(* IEC 61131-3 sources: json/test/String, 1 file *)

(* ---- TestJsonString.st ---- *)
USING AxUnit.Assert;
USING System.Strings;
USING Simatic.Ax.Conversion;

NAMESPACE Simatic.Ax.Json
    {TestFixture}
    CLASS TestJsonString

        VAR PROTECTED
            //e : JsonString := (value := 'value', key := 'test');
            e : JsonString := (value := 'my#1234,,,,', Key := 'test');
            expString, actString : STRING;
            cmpBuff : ARRAY[0..20] OF CHAR;
            doc : JsonDocument;
            buffer : ARRAY[0..200] OF CHAR;
        END_VAR

        {Test}
        METHOD PUBLIC TestSerialize_s_test_true
            VAR_TEMP
                len : DINT;
                res : BOOL;
            END_VAR
            doc.buffer := REF(buffer);
            e.Serialize(REF(doc));

            expString := '"test": "my#1234,,,,"';
            len := Strings.ToArray.OfCharCount(str := expString, arr := cmpBuff);
            res := CompareArray(first := buffer, scnd := cmpBuff, count := TO_INT(len));
            Equal(expected := TRUE, actual := res);

        END_METHOD

    END_CLASS
END_NAMESPACE
